// TIA Portal V17 export
// export: Created 2024-09-02T12:50:30.2979923Z, ExportSetting WithDefaults, DisplayName Totally Integrated Automation Portal, DisplayVersion V17, DisplayName TIA Portal Openness, DisplayVersion V17, DisplayName TIA Portal Version Control Interface, DisplayVersion V17, DisplayName STEP 7 Professional, DisplayVersion V17, DisplayName STEP 7 Safety, DisplayVersion V17, DisplayName WinCC Professional, DisplayVersion V17
TYPE "type_CognexDMOut"
// stored: IsFailsafeCompliant false
   STRUCT
      Ansteuerung { ExternalWritable := 'False'} : Struct   // Ansteuerung / Control
         Trigger_enable { ExternalWritable := 'False'} : Bool;   // Aufnamesteuerung: Trigger enable / Recording Status: Trigger enable
         Trigger { ExternalWritable := 'False'} : Bool;   // Aufnamesteuerung: Trigger / Recording Status: Trigger
         Res02 { ExternalWritable := 'False'} : Bool;   // Aufnamesteuerung: / Record control:
         Res03 { ExternalWritable := 'False'} : Bool;   // Aufnamesteuerung: / Record control:
         Res04 { ExternalWritable := 'False'} : Bool;   // Aufnamesteuerung: / Record control:
         Res05 { ExternalWritable := 'False'} : Bool;   // Aufnamesteuerung: / Record control:
         Res06 { ExternalWritable := 'False'} : Bool;   // Aufnamesteuerung: / Record control:
         Set_Offline { ExternalWritable := 'False'} : Bool;   // Aufnahmesteurung: Set offline / Recording status: Set offline
         Results_Buffer_Enable { ExternalWritable := 'False'} : Bool;   // Inspektionssteuerung: Buffer Results Enable / Inspection Control: Buffer Results Enable
         Results_Ack { ExternalWritable := 'False'} : Bool;   // Inspektionssteuerung: Inspection Results Acknowledge / Inspection Control: Inspection Results Acknowledge
         Res12 { ExternalWritable := 'False'} : Bool;   // Inspektionssteuerung: / Inspection control:
         Res13 { ExternalWritable := 'False'} : Bool;   // Inspektionssteuerung: / Inspection control:
         Res14 { ExternalWritable := 'False'} : Bool;   // Inspektionssteuerung: / Inspection control:
         Res15 { ExternalWritable := 'False'} : Bool;   // Inspektionssteuerung: / Inspection control:
         Res16 { ExternalWritable := 'False'} : Bool;   // Inspektionssteuerung: / Inspection control:
         Res17 { ExternalWritable := 'False'} : Bool;   // Inspektionssteuerung: / Inspection control:
         Set_Job_No { ExternalWritable := 'False'} : Byte;   // Parametersatz: Set Job Number / Parameter set: Set Job Number
         Softevent { ExternalWritable := 'False'} : Byte;   // Softevent / soft event
      END_STRUCT;
      Benutzerdaten { ExternalWritable := 'False'} : Struct   // Benutzerdaten (ab Byte 4) / User name (ab Byte 4)
         Option { ExternalWritable := 'False'} : Struct   // Option
            Data { ExternalWritable := 'False'} : Int;   // Kennung für die Ausführungsart des IBV-Systems / Identifier for the type of implementation of the IBV system
            Length { ExternalWritable := 'False'} : Int;   // Aktuelle Modis: TR-> Bildaufnahme und -auswertung durchführen / Current modes: TR-> Perform image acquisition and evaluation
         END_STRUCT;
         Data { ExternalWritable := 'False'} : Struct   // Date
            Data { ExternalWritable := 'False'} : Array[1..128] of Char;   // User Daten / User data
         END_STRUCT;
      END_STRUCT;
   END_STRUCT;
END_TYPE
